PROGRAM main
  VAR
    START_BUTTON : BOOL := FALSE;
    STOP_BUTTON : BOOL := FALSE;
    MOTOR_CONVEYER : BOOL := FALSE;
    CTU0 : CTU;
    SENSOR : BOOL := FALSE/STATE;
    reset : BOOL := FALSE;
    TON0 : TON;
    TON1 : TON;
    STATE : BOOL := FALSE;
  END_VAR

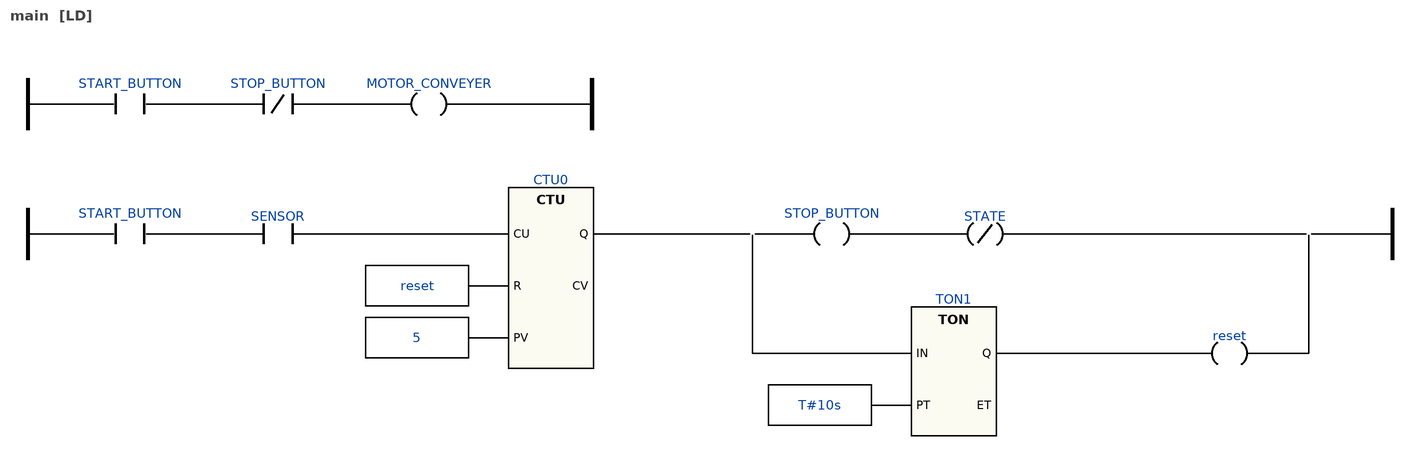
(* LD diagram, written out as Structured Text *)
MOTOR_CONVEYER := START_BUTTON AND NOT STOP_BUTTON;
CTU0(CU := START_BUTTON AND SENSOR, R := reset, PV := 5);
STOP_BUTTON := CTU0.Q;
STATE := NOT CTU0.Q;
TON1(IN := CTU0.Q, PT := T#10s);
reset := TON1.Q;
END_PROGRAM
